Staubli VAL3: SyncMovej.pjx

--- SyncMovej.pjx ---
Parameters version=s7.9 stackSize=5000 millimeterUnit=true
Program file=start.pgx
Program file=stop.pgx
Data file=SyncMovej.dtx

--- start.pgx ---
program start()
begin
  //利用4毫秒来实现同步功能














end
